TYPE ST_VCC :
STRUCT

(* Inputs *)
{attribute 'pytmc' := '
    pv: OPN_SW
	io: io
	'}
	pv_xOPN_SW	: BOOL;
	{attribute 'pytmc' := '
    pv:OVRD_OPN
	io: io
	'}
	xOvrdOpn	:	BOOL;
	{attribute 'pytmc' := '
    pv: OPN_OK
	io: i
	'}
	xOPN_OK	: BOOL;

(* Outputs *)
{attribute 'pytmc' := '
    pv: RUN_DO
	io: i
	'}
	q_xOPN_DO	: BOOL;

END_STRUCT
END_TYPE

(* stored: Version 1.1.0.1, ProductVersion 3.1.4020.12
   DUT ST_VCC: Id {29dc25c3-dd01-4b35-9336-905aa03d820f} *)
